PROGRAM MAIN
VAR
END_VAR

END_PROGRAM

(* stored: Version 1.1.0.1
   POU MAIN: Id {8a3569cd-6104-4581-88b5-3868e843a0c8} *)
